// TIA Portal V19 export
TYPE "PartCuttedBuffer_Item"
   STRUCT
      PTrkId : DInt;
      HeadCutPosition : LReal;
      TailCutPosition : LReal;
      R1_TailPosVirtPos : LReal;
      R2_TailPosVirtPos : LReal;
      Result : Int;   // 0=UNKNOW;1=GOOD;2=WRONG;3=TO CHECK
   END_STRUCT;
END_TYPE
